{attribute 'qualified_only'}
VAR_GLOBAL
	Start: BOOL;
	Stop: BOOL;
	Emergency: BOOL;
	Reset: BOOL;
END_VAR

(* stored: Version 1.1.0.1, ProductVersion 3.1.4024.4
   GVL AutoControlCommand: Id {22e194c5-4f63-4572-9b26-db34c6c7cf43} *)
